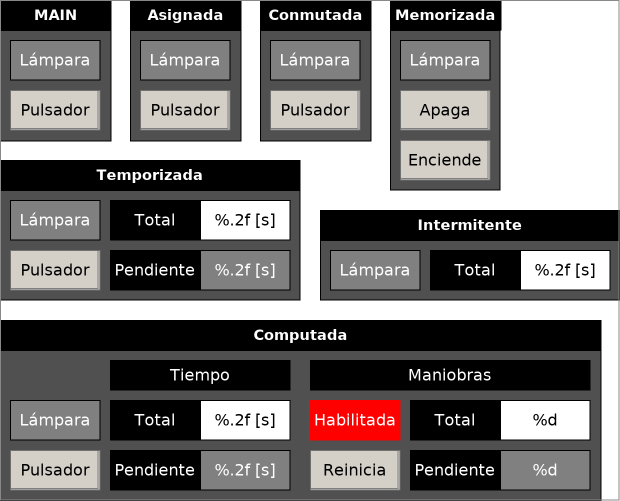
VISUALIZATION Visualization  // 620x501
    Rectangle (0,30 111x111)
    Rectangle (10,40 90x40), "Lámpara", colour toggle: MAIN.Lampara
    Button (10,90 90x40), "Pulsador"
        tap MAIN.Pulsador
    Rectangle (0,0 111x30), "MAIN"
    Rectangle (0,190 300x110)
    Rectangle (10,200 90x40), "Lámpara", colour toggle: MAIN.LamparaTemporizada.Lampara
    Button (10,250 90x40), "Pulsador"
        tap MAIN.LamparaTemporizada.Pulsador
    Rectangle (0,160 300x30), "Temporizada"
    Rectangle (110,200 90x40), "Total"
    Rectangle (200,200 90x40), "%.2f [s]", text variable: MAIN.LamparaTemporizada.TiempoEncendido
        OnMouseDown: write the text variable via Default
    Rectangle (110,250 90x40), "Pendiente"
    Rectangle (200,250 90x40), "%.2f [s]", text variable: MAIN.LamparaTemporizada.TiempoPendiente
    Rectangle (130,30 111x111)
    Rectangle (140,40 90x40), "Lámpara", colour toggle: MAIN.LamparaAsignada.Lampara
    Button (140,90 90x40), "Pulsador"
        tap MAIN.LamparaAsignada.Pulsador
    Rectangle (130,0 111x30), "Asignada"
    Rectangle (260,30 111x111)
    Rectangle (270,40 90x40), "Lámpara", colour toggle: MAIN.LamparaConmutada.Lampara
    Button (270,90 90x40), "Pulsador"
        tap MAIN.LamparaConmutada.Pulsador
    Rectangle (260,0 111x30), "Conmutada"
    Rectangle (0,350 601x151)
    Rectangle (10,400 90x40), "Lámpara", colour toggle: MAIN.LamparaComputada.Lampara
    Button (10,450 90x40), "Pulsador"
        tap MAIN.LamparaComputada.Pulsador
    Rectangle (0,320 601x30), "Computada"
    Rectangle (410,400 90x40), "Total"
    Rectangle (500,400 90x40), "%d", text variable: MAIN.LamparaComputada.ManiobrasTotales
        OnMouseDown: write the text variable via Default
    Rectangle (410,450 90x40), "Pendiente"
    Rectangle (500,450 90x40), "%d", text variable: MAIN.LamparaComputada.ManiobrasPendientes
    Button (310,450 90x40), "Reinicia"
        tap MAIN.LamparaComputada.Reinicia
    Rectangle (310,400 90x40), "Habilitada", colour toggle: MAIN.LamparaComputada.Habilitada
    Rectangle (110,400 90x40), "Total"
    Rectangle (200,400 90x40), "%.2f [s]", text variable: MAIN.LamparaComputada.TiempoEncendido
        OnMouseDown: write the text variable via Default
    Rectangle (110,450 90x40), "Pendiente"
    Rectangle (200,450 90x40), "%.2f [s]", text variable: MAIN.LamparaComputada.TiempoPendiente
    Rectangle (390,30 110x160)
    Rectangle (400,40 90x40), "Lámpara", colour toggle: MAIN.LamparaMemorizada.Lampara
    Button (400,90 90x40), "Apaga"
        tap MAIN.LamparaMemorizada.PulsadorDesconexion
    Rectangle (390,0 111x30), "Memorizada"
    Button (400,140 90x40), "Enciende"
        tap MAIN.LamparaMemorizada.PulsadorConexion
    Rectangle (110,360 180x30), "Tiempo"
    Rectangle (310,360 280x30), "Maniobras"
    Rectangle (320,240 300x60)
    Rectangle (330,250 90x40), "Lámpara", colour toggle: MAIN.LamparaIntermitente.Lampara
    Rectangle (320,210 300x30), "Intermitente"
    Rectangle (430,250 90x40), "Total"
    Rectangle (520,250 90x40), "%.2f [s]", text variable: MAIN.LamparaIntermitente.TiempoParpadeo
        OnMouseDown: write the text variable via Default
END_VISUALIZATION

(* stored: Version 1.1.0.1, ProductVersion 3.1.4024.15
   Visu Visualization: Id {9c96670d-5611-45f7-b475-36643b25dd97} *)
